TYPE TYP_HW_L4000_INSP_RESULTS :
STRUCT
	InspectionID AT %I* : UINT;
	InspectionResultCode AT %I* : UINT;
	Results AT %I* : ARRAY[0..63] OF BYTE;
END_STRUCT
END_TYPE

(* stored: Version 1.1.0.1, ProductVersion 3.1.4024.12
   DUT TYP_HW_L4000_INSP_RESULTS: Id {73c66c72-41b2-4884-b65e-0bb343f3a8cc} *)
